PROGRAM RecipeModule_R1
VAR
	shutDownFB:Shutdown;
	remainingTimeCalculator : RemainingTimeCalculator;
	
	DosingTick: INT;
	AbortTrig:R_Trig;
END_VAR
VAR_INPUT
	DosingTotalizerVolume: REAL;
END_VAR

IF R1.RecipeStep[0].Started AND R1.RecipeStep[0].StartedTime = '' THEN
	//Update StartedTime
	R1.RecipeStep[0].StartedTime := MAIN.concatenatedHourMinuteString;
END_IF

// Start Block and HC Mode Selection
IF R1.RecipeStep[R1.R1STEPS].Started THEN
  R1.R1STEPS:= R1.R1STEPS+1;
 // R1.AbortRecipe:=FALSE;
  R1.ClearRecipe:=FALSE;
  R1.RecipeEnded:=FALSE;
END_IF  
 
// Check Process or JACKET SELECTION
IF R1.RecipeStep[0].HeatCoolModeSelection THEN
	R1.HeatCoolTemperatureControlType:=TRUE;
	R1.TemperatureControl:=REAL_TO_DINT(R1.ReactorMassTemperature);
ELSE
	R1.HeatCoolTemperatureControlType:=FALSE;	
	R1.TemperatureControl:=REAL_TO_DINT(R1.JacketOutletTemperature);
END_IF

 IF R1.RecipeStep[R1.R1STEPS].HeatcoolEnabled THEN
	R1.HeatCoolSetPoint:=R1.RecipeStep[R1.R1STEPS].HeatCoolSetpointExpression;		
	R1.RecipeStep[R1.R1STEPS].HeatCoolStarted :=TRUE;
	IF R1.RecipeStep[R1.R1STEPS].HeatCoolStartedTime = '' THEN
		R1.RecipeStep[R1.R1STEPS].HeatCoolStartedTime := Main.concatenatedHourMinuteString;
	END_IF
	R1.HeatCoolStatus:=TRUE;
	
		///Check for condition in step  
	 IF ABS(R1.TemperatureControl-R1.RecipeStep[R1.R1STEPS].HeatCoolSetpointExpression )<0.5 THEN
		R1.RecipeStep[R1.R1STEPS].HeatcoolEnded :=TRUE;	
		IF R1.RecipeStep[R1.R1STEPS].HeatCoolEndedTime = '' THEN
			R1.RecipeStep[R1.R1STEPS].HeatCoolEndedTime := Main.concatenatedHourMinuteString;
		END_IF
	 END_IF     	
 END_IF
	
////Recipe block for stirrer
IF R1.RecipeStep[R1.R1STEPS].StirrerEnabled THEN
	R1.StirrerSetPoint:=R1.RecipeStep[R1.R1STEPS].StirrerSetPointExpression;
	R1.StirrerStatus:=TRUE;	
    R1.RecipeStep[R1.R1STEPS].StirrerStarted:=TRUE;
	IF R1.RecipeStep[R1.R1STEPS].StirrerStartedTime = '' THEN
		R1.RecipeStep[R1.R1STEPS].StirrerStartedTime := Main.concatenatedHourMinuteString;
	END_IF
	
	///Check the Actual speed to end the step
      IF ABS(R1.StirrerCurrentSpeed- R1.RecipeStep[R1.R1STEPS].StirrerSetPointExpression)<8 THEN
		R1.RecipeStep[R1.R1STEPS].StirrerEnded:=TRUE;
		IF R1.RecipeStep[R1.R1STEPS].StirrerEndedTime = '' THEN
			R1.RecipeStep[R1.R1STEPS].StirrerEndedTime := Main.concatenatedHourMinuteString;
		END_IF
	  END_IF
	//Check the rpm TO switch off the vfd
	  IF R1.RecipeStep[R1.R1STEPS].StirrerSetPointExpression=0 THEN
		R1.StirrerStatus:=FALSE;	
	  END_IF///
  END_IF 


(*////Wait Block*)
IF R1.RecipeStep[R1.R1STEPS].WaitEnabled AND NOT R1.RecipeStep[R1STEPS].WaitEnded THEN
    R1.RecipeStep[R1.R1STEPS].WaitStarted:=TRUE;
	IF R1.RecipeStep[R1.R1STEPS].WaitStartedTime = '' THEN
		R1.RecipeStep[R1.R1STEPS].WaitStartedTime := Main.concatenatedHourMinuteString;
	END_IF
	R1.WaitTick:=R1.WaitTick+1;
	IF R1.WaitTick=100  THEN
		//Update the Second Tick
		R1.WaitSecondTick:=R1.WaitSecondTick+1;
		R1.WaitTick:=0;
	END_IF
		
	IF  R1.WaitSecondTick=60  THEN
		//Update the Minute Tick
		R1.WaitMinuteTick:=R1.WaitMinuteTick+1;
		R1.WaitSecondTick:=0;
	END_IF	

	//Update the Remaining Time
	remainingTimeCalculator(elapsedSeconds:= R1.WaitSecondTick, elapsedMinutes:= R1.WaitMinuteTick, givenDuration:= DINT_TO_INT(R1.RecipeStep[R1.R1STEPS].WaitDuration), 
							leftOverSeconds=> R1.RecipeStep[R1.R1STEPS].WaitRemainingSeconds, leftOverMinutes=> R1.RecipeStep[R1.R1STEPS].WaitRemainingMinutes);
	R1.RecipeStep[R1.R1STEPS].WaitRemainingTime := INT_TO_STRING(R1.RecipeStep[R1.R1STEPS].WaitRemainingMinutes);
	R1.RecipeStep[R1.R1STEPS].WaitRemainingTime := CONCAT(STR1:= R1.RecipeStep[R1.R1STEPS].WaitRemainingTime, STR2:= ':');
	R1.RecipeStep[R1.R1STEPS].WaitRemainingTime := CONCAT(STR1:= R1.RecipeStep[R1.R1STEPS].WaitRemainingTime, STR2:= INT_TO_STRING(R1.RecipeStep[R1.R1STEPS].WaitRemainingSeconds));
	
	(*///To write ended time*)
	IF ABS(R1.WaitMinuteTick -R1.RecipeStep[R1.R1STEPS].WaitDuration)=0 THEN
		R1.RecipeStep[R1.R1STEPS].WaitEnded:=TRUE;
		IF R1.RecipeStep[R1.R1STEPS].WaitEndedTime = '' THEN
			R1.RecipeStep[R1.R1STEPS].WaitEndedTime := Main.concatenatedHourMinuteString;
		END_IF
		R1.WaitTick:=0;
		R1.WaitSecondTick:=0;
		R1.WaitMinuteTick:=0;
	END_IF
END_IF
	
IF R1.RecipeStep[R1STEPS].DosingEnabled AND NOT R1.RecipeStep[R1STEPS].DosingEnded THEN
	R1.RecipeStep[R1STEPS].DosingStarted := TRUE;
	IF R1.RecipeStep[R1.R1STEPS].DosingStartedTime = '' THEN
		R1.RecipeStep[R1.R1STEPS].DosingStartedTime := Main.concatenatedHourMinuteString;
	END_IF
	//Update Totalized Volume
		IF  R1.DosingPumpStatus_1 THEN
			DosingTick:=DosingTick+1;
		END_IF
		   
	  IF DosingTick=100 THEN
		  DosingTotalizerVolume:=DosingTotalizerVolume+(R1.RecipeStep[R1STEPS].DosingRateSetpointExpression/2.7 * 0.045);	  
	  END_IF
	  
	  IF DosingTick>100 THEN
		  DosingTick:=0;
	  END_IF
	  
	IF DosingTotalizerVolume < R1.RecipeStep[R1STEPS].DosingMaxAmount THEN
		IF R1.DosingPumpStatus_1 THEN
			IF R1.TemperatureControl < R1.RecipeStep[R1STEPS].DosingStopTemp THEN
				R1.DosingPumpStatus_1 := TRUE;
				R1.DosingPumpSetPoint_1 := R1.RecipeStep[R1STEPS].DosingRateSetpointExpression;
			ELSE
				R1.DosingPumpStatus_1 := FALSE;
				R1.DosingPumpSetPoint_1 := 0;
			END_IF
		ELSE
			IF DosingTotalizerVolume = 0 AND R1.TemperatureControl > R1.RecipeStep[R1STEPS].DosingResumeTemp AND R1.TemperatureControl < R1.RecipeStep[R1STEPS].DosingStopTemp THEN
				//Logic for starting Dosing Pump First Time in a Recipe Step
				R1.DosingPumpStatus_1 := TRUE;
				R1.DosingPumpSetPoint_1 := R1.RecipeStep[R1STEPS].DosingRateSetpointExpression;
			END_IF
			
			IF R1.TemperatureControl < R1.RecipeStep[R1STEPS].DosingResumeTemp THEN
				R1.DosingPumpStatus_1 := TRUE;
				R1.DosingPumpSetPoint_1 := R1.RecipeStep[R1STEPS].DosingRateSetpointExpression;
			END_IF
		END_IF
	ELSE
		R1.DosingPumpStatus_1 := FALSE;
		R1.DosingPumpSetPoint_1 := 0;
		R1.RecipeStep[R1STEPS].DosingEnded := TRUE;
		IF R1.RecipeStep[R1.R1STEPS].DosingEndedTime = '' THEN
			R1.RecipeStep[R1.R1STEPS].DosingEndedTime := Main.concatenatedHourMinuteString;
		END_IF
		DosingTick := 0;
		DosingTotalizerVolume:=0;
	END_IF
END_IF

IF R1.R1STEPS>0 THEN 

(*//Step control block To increment to next step*)
 R1.TotalEnabledValue:=BOOL_TO_INT(R1.RecipeStep[R1.R1STEPS].HeatcoolEnabled)+BOOL_TO_INT(R1.RecipeStep[R1.R1STEPS].StirrerEnabled)+BOOL_TO_INT(R1.RecipeStep[R1.R1STEPS].WaitEnabled)+BOOL_TO_INT( R1.RecipeStep[R1.R1STEPS].DosingEnabled);
 R1.TotalEndedValue:=BOOL_TO_INT(R1.RecipeStep[R1.R1STEPS].HeatCoolEnded)+BOOL_TO_INT(R1.RecipeStep[R1.R1STEPS].StirrerEnded)+BOOL_TO_INT(R1.RecipeStep[R1.R1STEPS].WaitEnded)+BOOL_TO_INT( R1.RecipeStep[R1.R1STEPS].DosingEnded);

    IF (R1.TotalEnabledValue - R1.TotalEndedValue)=0 THEN 
		R1.R1STEPS:=R1.R1STEPS+1;
    END_IF
END_IF
  
 (* ///To End the Recipe**)
 IF  R1.NumberOfRecipeSteps = R1.R1STEPS THEN
	 R1.StirrerStatus:=FALSE;
	 R1.StirrerSetPoint:=0;
	 R1.HeatCoolStatus:=FALSE;
	 R1.HeatCoolSetPoint:=0;	
     R1.StepCompleted:=FALSE;	 
	 R1.RecipeEnded:=TRUE;
	 R1.RecipeStatus:=FALSE;
 END_IF
  
(* //TO ABORT RECIPE*)
AbortTrig(CLK:=R1.AbortRecipe,Q=>);
IF AbortTrig.Q THEN
	shutDownFB(GvlIdentifier := 'R1');
	AbortTrig.CLK := FALSE;
END_IF

END_PROGRAM

(* stored: Version 1.1.0.1, ProductVersion 3.1.4024.0
   POU RecipeModule_R1: Id {416c4a34-82f5-4d2d-8905-a8547ed16d93}, SpecialFunc None *)
